Omron CX-Programmer project NewProject (CX-Programmer 9.75)

# PLC TankLevel: CJ2M CPU11

## Program NewProgram1 (cyclic task 0)
Local symbols
IV1 100.02 BOOL
M1 100.01 BOOL
MainSupply 100.00 BOOL
Motor 100.00 BOOL
OVL 100.03 BOOL
Start 0.00 BOOL
Stop 0.01 BOOL
Sw1 0.02 BOOL
Sw2 0.03 BOOL
Sw3 0.05 BOOL
Sw4 0.06 BOOL

### Section Section1

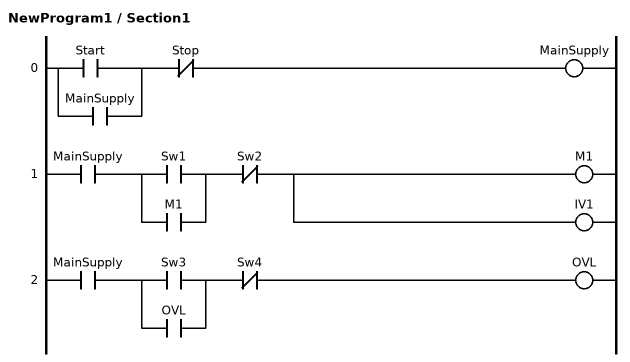
; rung 0
LD Start
OR MainSupply
ANDNOT Stop
OUT MainSupply
; rung 1
LD MainSupply
LD Sw1
OR M1
ANDLD
ANDNOT Sw2
OUT M1
OUT IV1
; rung 2
LD MainSupply
LD Sw3
OR OVL
ANDLD
ANDNOT Sw4
OUT OVL

### Section END
; rung 0
END(001)